FUNCTION_BLOCK FB_HE_SATT_FilterCombinationToTransmissionTestDouble IMPLEMENTS I_HE_SATT_FilterCombinationToTransmission
VAR CONSTANT
    nMaxIndex : INT := 10;
END_VAR
VAR
    afMinimumTransmissionResultSequence : ARRAY[1..nMaxIndex] OF LREAL;
    afMaximumTransmissionResultSequence : ARRAY[1..nMaxIndex] OF LREAL;
    nIndexForNextAdditionToSequence : INT;
    nIndexInSequence : INT;
END_VAR


METHOD CalculateTransmission
VAR_INPUT
	fPhotonEnergy_eV	: LREAL;
	iFilterCombination	: I_HE_SATT_FilterCombination;
END_VAR
VAR_OUTPUT
	fMinimumTransmission	: LREAL;
	fMaximumTransmission	: LREAL;
END_VAR

THIS^.nIndexInSequence := THIS^.nIndexInSequence + 1;

fMinimumTransmission := THIS^.afMinimumTransmissionResultSequence[THIS^.nIndexInSequence];
fMaximumTransmission := THIS^.afMaximumTransmissionResultSequence[THIS^.nIndexInSequence];

IF THIS^.nIndexInSequence > THIS^.nMaxIndex THEN
    THIS^.nIndexInSequence := 0;
END_IF
END_METHOD


METHOD PUBLIC PushTransmissionResultToSequence
VAR_INPUT
    fMinimumTransmission : LREAL;
    fMaximumTransmission : LREAL;
END_VAR

THIS^.nIndexForNextAdditionToSequence := THIS^.nIndexForNextAdditionToSequence + 1;

THIS^.afMinimumTransmissionResultSequence[THIS^.nIndexForNextAdditionToSequence] := fMinimumTransmission;
THIS^.afMaximumTransmissionResultSequence[THIS^.nIndexForNextAdditionToSequence] := fMaximumTransmission;
END_METHOD


METHOD PUBLIC Reset

THIS^.nIndexInSequence := 0;
END_METHOD

END_FUNCTION_BLOCK

(* stored: Version 1.1.0.1
   POU FB_HE_SATT_FilterCombinationToTransmissionTestDouble: Id {dc6cd939-bb8c-4dbc-bad7-09e38e5b1ec5}, SpecialFunc None
   Method CalculateTransmission: Id {484901a1-185b-4414-9811-81a366f92c86}
   Method PushTransmissionResultToSequence: Id {1f6ee084-b2de-4f4d-9335-e238d0c71420}
   Method Reset: Id {b677cfd8-c9af-4497-aaf7-a7583ef609b2} *)
